TYPE ST_StewartControl :
STRUCT
	eta: ARRAY[0..5] OF LREAL;
END_STRUCT
END_TYPE

(* stored: Version 1.1.0.1, ProductVersion 3.1.4022.7
   DUT ST_StewartControl: Id {bd0ca14b-317a-4883-81d9-ee36e7babaa4} *)
